// TIA Portal V17 export
// export: Created 2025-03-05T08:01:02.9893917Z, ExportSetting WithDefaults, DisplayName Totally Integrated Automation Portal, DisplayVersion V17 Update 8, DisplayName TIA Portal Openness, DisplayVersion V17 Update 8, DisplayName TIA Portal Version Control Interface, DisplayVersion V17, DisplayName SINAMICS Startdrive Advanced, DisplayVersion V17 SP2, DisplayName SINAMICS Startdrive G110M, G120, G120C, G120D, G120P, G115D, DisplayVersion V17 SP2, DisplayName SINAMICS Startdrive G130, G150, S120, S150, SINAMICS MV, S210, DisplayVersion V17 SP2, DisplayName STEP 7 Professional, DisplayVersion V17 Update 8, DisplayName SINUMERIK ONE STEP 7 Toolbox, DisplayVersion V17 Update 12, DisplayName SINUMERIK 840D sl STEP 7 Toolbox, DisplayVersion V17 Update 12, DisplayName STEP 7 Safety, DisplayVersion V17 Update 6, DisplayName WinCC Advanced, DisplayVersion V17 Update 8
DATA_BLOCK "LTLP_ToolLifeTimeDB"   // DB521
{ DB_Accessible_From_OPC_UA := 'FALSE' }
// stored: AutoNumber true, DBAccessibleFromOPCUA false, DBAccessibleFromWebserver true, InstanceOfName LTLP_ToolLifeTime, InstanceOfType FB
"LTLP_ToolLifeTime"
   // VAR_OUTPUT
   //    ERROR : Word;
   // END_VAR
   // VAR_IN_OUT
   //    TOOL_COUNT : Variant;
   //    TOOL_STATE : Variant;
   //    HMI_DB : "LTLP_typeHmiProInterface";
   // END_VAR
   // VAR
   //    countOfWkzCount : Int;
   //    countOfWkzState : Int;
   //    impulsCount : Array[1..96] of Bool;
   //    triggerCount : Array[1..96] of Bool;
   //    wkzCount { ExternalAccessible := 'False'; ExternalVisible := 'False'; ExternalWritable := 'False'} : Array[1..96] of Bool;
   //    wkzState { ExternalAccessible := 'False'; ExternalVisible := 'False'; ExternalWritable := 'False'} : Array[1..96] of Byte;
   // END_VAR
BEGIN
END_DATA_BLOCK
